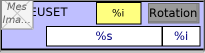
VISUALIZATION VISU_CREUSET_V3  // 205x53
VAR_IN_OUT
	m_Input_CREUSET : BLOCK_IND_CR_379_TELEMARK_V3;
END_VAR
    Rectangle (0,0 205x50)
    RoundedRectangle (96,2 45x22), "%i", text variable: m_Input_CREUSET.PRM_NCR, invisible if: NOT Global_Variables.PRG_USER.ACTU_USER.MAINTENANCE OR NOT MACHINE.State_manu
        OnMouseDown: write the text variable via InputWithLimits
    Rectangle (0,3 81x18), "CREUSET"
    Rectangle (1,26 48x18), text list: 'TextList_Evap', text index: 5
    RoundedRectangle (46,26 116x20), "%s", text variable: m_Input_CREUSET.STATE_MAT
    RoundedRectangle (162,26 38x20), "%i", text variable: m_Input_CREUSET.STATE_POS
    Button (148,3 51x20), "Rotation", invisible if: NOT m_Input_CREUSET.AUTOR_Change_IHM OR NOT PRG_User.ACTU_USER.MAINTENANCE
        tap m_Input_CREUSET.M_Change
    Image (1,-3 32x32), invisible if: NOT m_Input_CREUSET.State_nok, image: MesImages.warning
END_VISUALIZATION

(* stored: Version 1.1.0.1, ProductVersion 3.1.4026.18
   Visu VISU_CREUSET_V3: Id {c45edcef-8f94-416f-ad7e-324adb838685} *)
